# EPICS substitutions: mc05/tpmacApp/Db/encRead.substitutions
file "db/encRead.db"
{
pattern
{MtrName,              				N,	MRES}
{"XF:16IDB-OP{Fltr:Atn-Ax:X1}Mtr_",		5,	0.000625}
{"XF:16IDB-OP{Fltr:Atn-Ax:X2}Mtr_",		6,      0.000625}
{"XF:16IDB-OP{Fltr:Atn-Ax:X3}Mtr_",		7,      0.000625}
}
